PROGRAM POU
VAR
END_VAR

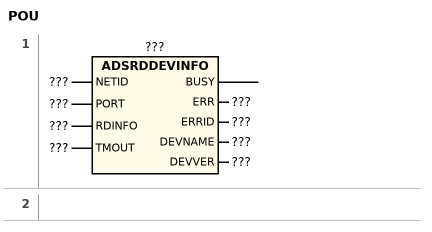
// NETWORK 1
???(); // ADSRDDEVINFO

// NETWORK 2

END_PROGRAM

(* stored: Version 1.1.0.1, ProductVersion 3.1.4024.12
   POU POU: Id {5e6affda-a3fc-4079-af85-42f6eb2d9529}, SpecialFunc None *)
